Universal Robots PolyScope program: OperacionAtornilladoFinal.urp

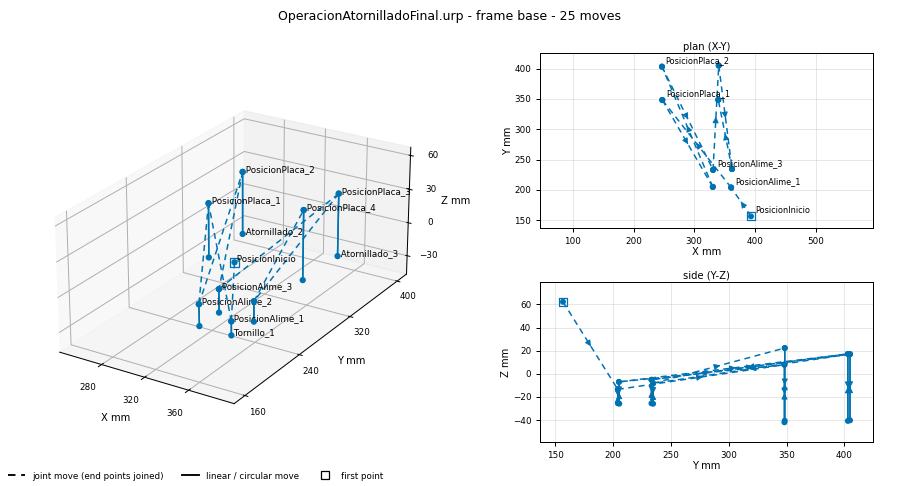
[picture p0: tool path of OperacionAtornilladoFinal.urp in frame base, 25 of 25 moves have a stored position in this frame; points joined in program order, loops and branches not executed]
Program OperacionAtornilladoB (installation=default directory=/programs/usbdisk createdIn=3.1.17195.0 lastSavedIn=3.15.6.106324 robotSerialNumber=2019330210)
Calibrated DH parameters: a=[0.000083, -0.175866, -0.153432, 0.0001, -0.000098, 0]; d=[0.152081, -62.187483, 140.989097, -78.689592, 0.085174, 0.082372]; alpha=[1.571415, -0.00271, -0.001881, 1.57151, -1.571414, 0]; deltaTheta=[-0.000402, 0.764772, -1.531542, 0.76907, -0.000461, 0.000675]
Robot Program (runOnlyOnce=true)
  MoveJ speed 60 deg/s, acceleration 80 deg/s^2 (useActiveTCP=false)
    Waypoint PosicionInicio: TCP in base x=393.541 y=156.505 z=62.302 mm, rx=-3.0249 ry=0.8416 rz=0.0079 rad; joints [36.821, -125.525, -85.808, -58.858, 90.277, -22.054] deg; flange x=393.956 y=156.214 z=157.301 mm, rx=-3.0249 ry=0.8416 rz=0.0079 rad
  PiezaPreparada :=  (valueSource=Operator message=Esta lista la pieza de trabajo y los tornillo? valueType=Boolean)
  Wait Condition expression=PiezaPreparada≟ True
  Script: write_port_register(128,4)
  Script: write_port_register(129,0)
  'Ingresar el paso del tornillo en (mm)'
  PasoTornillo :=  (valueSource=Operator message=Ingresar paso en (mm) valueType=Float)
  'Ingresar longitud roscada en (mm)'
  LongitudRoscada :=  (valueSource=Operator message=Longitud roscada en (mm) valueType=Float)
  'Ingresar velocidad de roscado en grados'
  VelocidadRoscar :=  (valueSource=Operator message=Velocidad de roscado en (deg/sec) valueType=Integer)
  'Calcula el tiempo de operacion de funcion speedj'
  TiempoRoscado := LongitudRoscada/((PasoTornillo/360)*VelocidadRoscar)
  'Convierte la velocidad a radianes'
  VelocidadRoscar := d2r(VelocidadRoscar)
  'Ciclo primer tornillo'
  MoveJ speed 60 deg/s, acceleration 80 deg/s^2 (useActiveTCP=false)
    Waypoint PosicionAlime_1: TCP in base x=360.784 y=203.988 z=-13.476 mm, rx=-3.025 ry=0.8415 rz=0.0081 rad; joints [44.95, -135.259, -93.311, -41.584, 90.299, -13.931] deg; flange x=361.213 y=203.695 z=81.523 mm, rx=-3.025 ry=0.8415 rz=0.0081 rad
  MoveL speed 250 mm/s, acceleration 1200 mm/s^2 (useActiveTCP=false) feature=Base
    Waypoint Tornillo_1: TCP in base x=360.82 y=204.003 z=-25.508 mm, rx=-3.0248 ry=0.8417 rz=0.0081 rad; joints [44.947, -137.423, -93.379, -39.347, 90.299, -13.926] deg; flange x=361.243 y=203.703 z=69.491 mm, rx=-3.0248 ry=0.8417 rz=0.0081 rad
  MoveL speed 250 mm/s, acceleration 1200 mm/s^2 (useActiveTCP=false) feature=Base
    Waypoint PosicionAlime_1: TCP in base x=360.784 y=203.988 z=-13.476 mm, rx=-3.025 ry=0.8415 rz=0.0081 rad; joints [44.95, -135.259, -93.311, -41.584, 90.299, -13.931] deg; flange x=361.213 y=203.695 z=81.523 mm, rx=-3.025 ry=0.8415 rz=0.0081 rad
  Script: write_port_register(128,3)
  MoveJ speed 60 deg/s, acceleration 80 deg/s^2 (useActiveTCP=false)
    Waypoint PosicionPlaca_1: TCP in base x=247.457 y=348.17 z=7.856 mm, rx=-3.0249 ry=0.8418 rz=0.0081 rad; joints [69.593, -133.835, -88.282, -47.904, 90.285, 10.723] deg; flange x=247.883 y=347.879 z=102.855 mm, rx=-3.0249 ry=0.8418 rz=0.0081 rad
  MoveL speed 250 mm/s, acceleration 1200 mm/s^2 (useActiveTCP=false) feature=Base
    Waypoint Atornillado_1: TCP in base x=247.407 y=348.174 z=-41.976 mm, rx=-3.025 ry=0.8416 rz=0.0081 rad; joints [69.595, -142.346, -88.725, -38.954, 90.282, 10.714] deg; flange x=247.839 y=347.888 z=53.022 mm, rx=-3.025 ry=0.8416 rz=0.0081 rad
  Force Frame feature=Base; selection=[0, 0, 1, 0, 0, 0]; wrench=[0, 0, -20, 0, 0, 0]; limitsForce=[0.15, 0.15, 0.15, 1.047198, 1.047198, 1.047198]; limitsMotion=[0.1, 0.1, 0.1, 0.349066, 0.349066, 0.349066]
    Script: speedj([0,0,0,0,0,VelocidadRoscar],6.28,TiempoRoscado)
  'Reinicia el conteo de giros'
  Script: reset_revolution_counter()
  MoveL speed 250 mm/s, acceleration 1200 mm/s^2 (useActiveTCP=false) feature=Base
    Waypoint PosicionPlaca_1: TCP in base x=247.457 y=348.17 z=7.856 mm, rx=-3.0249 ry=0.8418 rz=0.0081 rad; joints [69.593, -133.835, -88.282, -47.904, 90.285, 10.723] deg; flange x=247.883 y=347.879 z=102.855 mm, rx=-3.0249 ry=0.8418 rz=0.0081 rad
  Script: write_port_register(129,1)
  'Ciclo segundo tornillo'
  MoveJ speed 60 deg/s, acceleration 80 deg/s^2 (useActiveTCP=false)
    Waypoint PosicionAlime_2: TCP in base x=330.564 y=204.94 z=-6.993 mm, rx=3.0177 ry=-0.8594 rz=0.0081 rad; joints [48.637, -129.963, -102.293, -37.915, 89.649, -9.544] deg; flange x=330.192 y=205.432 z=88.005 mm, rx=3.0177 ry=-0.8594 rz=0.0081 rad
  MoveL speed 250 mm/s, acceleration 1200 mm/s^2 (useActiveTCP=false) feature=Base
    Waypoint Tornillo_2: TCP in base x=330.739 y=205.241 z=-25.856 mm, rx=3.0194 ry=-0.8597 rz=0.0093 rad; joints [48.642, -133.673, -102.485, -33.904, 89.653, -9.544] deg; flange x=330.256 y=205.59 z=69.142 mm, rx=3.0194 ry=-0.8597 rz=0.0093 rad
  MoveL speed 250 mm/s, acceleration 1200 mm/s^2 (useActiveTCP=false) feature=Base
    Waypoint PosicionAlime_2: TCP in base x=330.564 y=204.94 z=-6.993 mm, rx=3.0177 ry=-0.8594 rz=0.0081 rad; joints [48.637, -129.963, -102.293, -37.915, 89.649, -9.544] deg; flange x=330.192 y=205.432 z=88.005 mm, rx=3.0177 ry=-0.8594 rz=0.0081 rad
  Script: write_port_register(128,2)
  MoveJ speed 60 deg/s, acceleration 80 deg/s^2 (useActiveTCP=false)
    Waypoint PosicionPlaca_2: TCP in base x=246.928 y=403.056 z=17.21 mm, rx=3.0176 ry=-0.8592 rz=0.008 rad; joints [72.251, -141.613, -69.05, -59.655, 89.643, 14.068] deg; flange x=246.568 y=403.556 z=112.208 mm, rx=3.0176 ry=-0.8592 rz=0.008 rad
  MoveL speed 250 mm/s, acceleration 1200 mm/s^2 (useActiveTCP=false) feature=Base
    Waypoint Atornillado_2: TCP in base x=246.947 y=403.084 z=-40.761 mm, rx=3.0177 ry=-0.8593 rz=0.008 rad; joints [72.248, -150.032, -69.983, -50.295, 89.636, 14.057] deg; flange x=246.579 y=403.573 z=54.237 mm, rx=3.0177 ry=-0.8593 rz=0.008 rad
  Force Frame feature=Base; selection=[0, 0, 1, 0, 0, 0]; wrench=[0, 0, -20, 0, 0, 0]; limitsForce=[0.15, 0.15, 0.15, 1.047198, 1.047198, 1.047198]; limitsMotion=[0.1, 0.1, 0.1, 0.349066, 0.349066, 0.349066]
    Script: speedj([0,0,0,0,0,VelocidadRoscar],6.28,TiempoRoscado)
  Script: reset_revolution_counter()
  MoveL speed 250 mm/s, acceleration 1200 mm/s^2 (useActiveTCP=false) feature=Base
    Waypoint PosicionPlaca_2: TCP in base x=246.928 y=403.056 z=17.21 mm, rx=3.0176 ry=-0.8592 rz=0.008 rad; joints [72.251, -141.613, -69.05, -59.655, 89.643, 14.068] deg; flange x=246.568 y=403.556 z=112.208 mm, rx=3.0176 ry=-0.8592 rz=0.008 rad
  Script: write_port_register(129,2)
  'Ciclo tercer tornillo'
  MoveJ speed 60 deg/s, acceleration 80 deg/s^2 (useActiveTCP=false)
    Waypoint PosicionAlime_3: TCP in base x=331.009 y=233.108 z=-5.144 mm, rx=-3.0122 ry=0.8585 rz=-0.0157 rad; joints [51.288, -131.979, -97.603, -39.795, 89.682, -6.87] deg; flange x=329.848 y=232.508 z=89.847 mm, rx=-3.0122 ry=0.8585 rz=-0.0157 rad
  MoveL speed 250 mm/s, acceleration 1200 mm/s^2 (useActiveTCP=false) feature=Base
    Waypoint Tornillo_3: TCP in base x=331.033 y=233.085 z=-25.535 mm, rx=-3.0121 ry=0.8587 rz=-0.0157 rad; joints [51.281, -135.766, -97.802, -35.805, 89.681, -6.87] deg; flange x=329.87 y=232.479 z=69.456 mm, rx=-3.0121 ry=0.8587 rz=-0.0157 rad
  MoveL speed 250 mm/s, acceleration 1200 mm/s^2 (useActiveTCP=false) feature=Base
    Waypoint PosicionAlime_3: TCP in base x=331.009 y=233.108 z=-5.144 mm, rx=-3.0122 ry=0.8585 rz=-0.0157 rad; joints [51.288, -131.979, -97.603, -39.795, 89.682, -6.87] deg; flange x=329.848 y=232.508 z=89.847 mm, rx=-3.0122 ry=0.8585 rz=-0.0157 rad
  Script: write_port_register(128,1)
  MoveJ speed 60 deg/s, acceleration 80 deg/s^2 (useActiveTCP=false)
    Waypoint PosicionPlaca_3: TCP in base x=340.417 y=404.94 z=17.033 mm, rx=-3.0122 ry=0.8587 rz=-0.0155 rad; joints [62.253, -156.618, -38.492, -74.35, 89.428, 4.102] deg; flange x=339.268 y=404.35 z=112.025 mm, rx=-3.0122 ry=0.8587 rz=-0.0155 rad
  MoveL speed 250 mm/s, acceleration 1200 mm/s^2 (useActiveTCP=false) feature=Base
    Waypoint Atornillado_3: TCP in base x=340.447 y=404.922 z=-40.234 mm, rx=-3.0123 ry=0.8587 rz=-0.0157 rad; joints [62.25, -163.651, -39.758, -66.049, 89.419, 4.081] deg; flange x=339.288 y=404.334 z=54.757 mm, rx=-3.0123 ry=0.8587 rz=-0.0157 rad
  Force Frame feature=Base; selection=[0, 0, 1, 0, 0, 0]; wrench=[0, 0, -20, 0, 0, 0]; limitsForce=[0.15, 0.15, 0.15, 1.047198, 1.047198, 1.047198]; limitsMotion=[0.1, 0.1, 0.1, 0.349066, 0.349066, 0.349066]
    Script: speedj([0,0,0,0,0,VelocidadRoscar],6.28,TiempoRoscado)
  Script: reset_revolution_counter()
  MoveL speed 250 mm/s, acceleration 1200 mm/s^2 (useActiveTCP=false) feature=Base
    Waypoint PosicionPlaca_3: TCP in base x=340.417 y=404.94 z=17.033 mm, rx=-3.0122 ry=0.8587 rz=-0.0155 rad; joints [62.253, -156.618, -38.492, -74.35, 89.428, 4.102] deg; flange x=339.268 y=404.35 z=112.025 mm, rx=-3.0122 ry=0.8587 rz=-0.0155 rad
  Script: write_port_register(129,3)
  'Ciclo cuarto tornillo'
  MoveJ speed 60 deg/s, acceleration 80 deg/s^2 (useActiveTCP=false)
    Waypoint PosicionAlime_4: TCP in base x=362.333 y=234.536 z=-8.263 mm, rx=-3.0119 ry=0.8584 rz=-0.0159 rad; joints [47.996, -136.959, -88.001, -44.381, 89.704, -10.164] deg; flange x=361.155 y=233.912 z=86.727 mm, rx=-3.0119 ry=0.8584 rz=-0.0159 rad
  MoveL speed 250 mm/s, acceleration 1200 mm/s^2 (useActiveTCP=false) feature=Base
    Waypoint Tornillo_4: TCP in base x=362.3 y=234.482 z=-25.908 mm, rx=-3.0121 ry=0.8585 rz=-0.0159 rad; joints [47.996, -139.961, -88.148, -41.243, 89.695, -10.162] deg; flange x=361.126 y=233.879 z=69.083 mm, rx=-3.0121 ry=0.8585 rz=-0.0159 rad
  MoveL speed 250 mm/s, acceleration 1200 mm/s^2 (useActiveTCP=false) feature=Base
    Waypoint PosicionAlime_4: TCP in base x=362.333 y=234.536 z=-8.263 mm, rx=-3.0119 ry=0.8584 rz=-0.0159 rad; joints [47.996, -136.959, -88.001, -44.381, 89.704, -10.164] deg; flange x=361.155 y=233.912 z=86.727 mm, rx=-3.0119 ry=0.8584 rz=-0.0159 rad
  Script: write_port_register(128,0)
  MoveJ speed 60 deg/s, acceleration 80 deg/s^2 (useActiveTCP=false)
    Waypoint PosicionPlaca_4: TCP in base x=339.597 y=348.447 z=22.318 mm, rx=-3.0121 ry=0.8586 rz=-0.0157 rad; joints [59.124, -143.713, -63.611, -62.099, 89.514, 0.971] deg; flange x=338.433 y=347.842 z=117.309 mm, rx=-3.0121 ry=0.8586 rz=-0.0157 rad
  MoveL speed 250 mm/s, acceleration 1200 mm/s^2 (useActiveTCP=false) feature=Base
    Waypoint Atornillado_4: TCP in base x=339.568 y=348.412 z=-40.605 mm, rx=-3.0123 ry=0.8585 rz=-0.0157 rad; joints [59.123, -152.487, -64.776, -52.171, 89.509, 0.954] deg; flange x=338.412 y=347.822 z=54.386 mm, rx=-3.0123 ry=0.8585 rz=-0.0157 rad
  Force Frame feature=Base; selection=[0, 0, 1, 0, 0, 0]; wrench=[0, 0, -20, 0, 0, 0]; limitsForce=[0.15, 0.15, 0.15, 1.047198, 1.047198, 1.047198]; limitsMotion=[0.1, 0.1, 0.1, 0.349066, 0.349066, 0.349066]
    Script: speedj([0,0,0,0,0,VelocidadRoscar],6.28,TiempoRoscado)
  Script: reset_revolution_counter()
  MoveL speed 250 mm/s, acceleration 1200 mm/s^2 (useActiveTCP=false) feature=Base
    Waypoint PosicionPlaca_4: TCP in base x=339.597 y=348.447 z=22.318 mm, rx=-3.0121 ry=0.8586 rz=-0.0157 rad; joints [59.124, -143.713, -63.611, -62.099, 89.514, 0.971] deg; flange x=338.433 y=347.842 z=117.309 mm, rx=-3.0121 ry=0.8586 rz=-0.0157 rad
  Script: write_port_register(129,4)
  'Final de operacion'
